PROGRAM MAINFast
VAR
	test : BOOL;
END_VAR

test := NOT test;

END_PROGRAM

(* stored: Version 1.1.0.1
   POU MAINFast: Id {3d6956bb-1f86-48d0-b4c5-87dad5ac6c11}, SpecialFunc None *)
